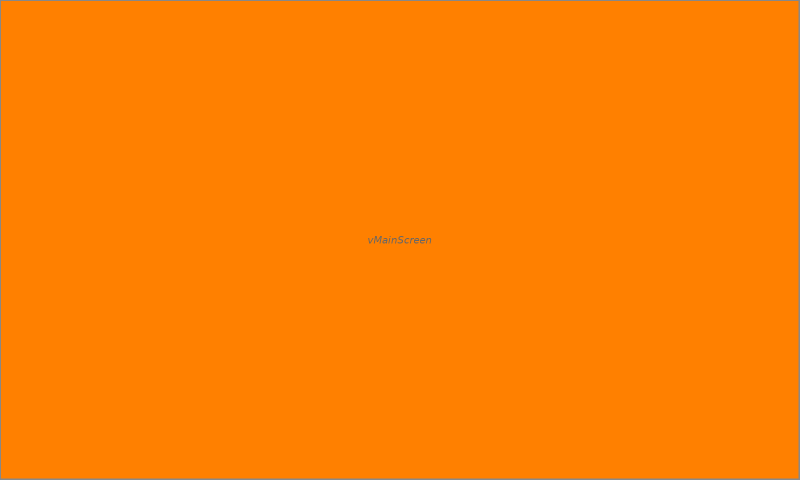
VISUALIZATION vMain  // 800x480
    Frame (0,0 800x480)
        shows vMainScreen(arChamber := MAIN.fb.arFbChamber, arParams := GVL_TesterParams.arstParams, arControl := GVL_TesterParams.arstControl, arTestParams := GVL_TesterParams.arTestParams)
END_VISUALIZATION

(* stored: Version 1.1.0.1, ProductVersion 3.1.4024.12
   Visu vMain: Id {8f3bb27e-2c8f-4987-943b-11137d390dae} *)
